// TIA Portal V20 export
DATA_BLOCK "DB_Manual"   // DB22
// stored: Access Published, MemoryReserve 100, Namespace Global
   VAR
      Conveyor : Struct
         ID : Int;
         Enable : Bool;
         Run : Bool;
         in : Bool;
      END_STRUCT;
      Line : Struct
         A1 : Struct
            Conveyor { S7_SetPoint := 'True'} : Array[_.gMinA1.._.gMaxA1] of "Global.ManualInputs";
         END_STRUCT;
         B1 : Struct
            Conveyor { S7_SetPoint := 'True'} : Array[_.gMinB1.._.gMaxB1] of "Global.ManualInputs";
         END_STRUCT;
         C1 : Struct
            Conveyor { S7_SetPoint := 'True'} : Array[_.gMinC1.._.gMaxC1] of "Global.ManualInputs";
         END_STRUCT;
         D1 : Struct
            Conveyor { S7_SetPoint := 'True'} : Array[_.gMinD1.._.gMaxD1] of "Global.ManualInputs";
         END_STRUCT;
      END_STRUCT;
   END_VAR
BEGIN
END_DATA_BLOCK
